TYPE E_AteqEndianType :
(
	LittleEndian,	// EthernetIP
	BigEndian		// Profinet
);
END_TYPE

(* stored: Version 1.1.0.1
   DUT E_AteqEndianType: Id {8c6a36e8-f33d-428b-b83a-481b140c04eb} *)
